// Mitsubishi GX Developer project: Пресс 70 крышка(алгоритм аварии при невыбросе крышки)   PLC: Q04UDEH

PROGRAM MAIN
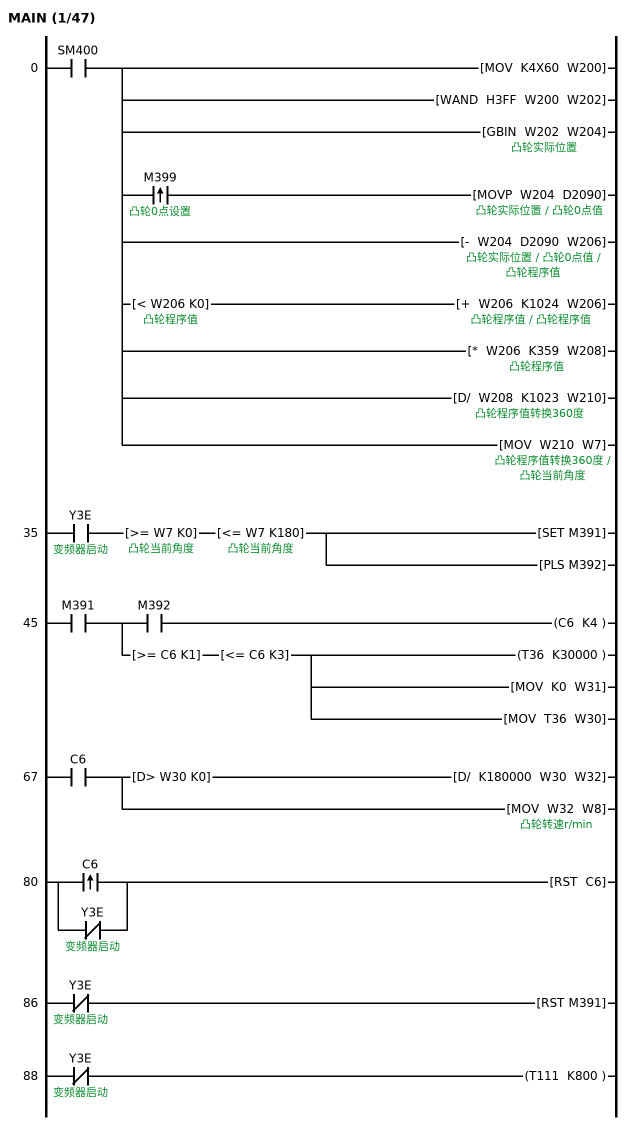
0     LD      SM400
      MOV     K4X60 W200  ; 绝地值编码器1
      WAND    H3FF W200 W202
      GBIN    W202 W204  ; 凸轮实际位置
      MPS
      ANDP    M399  ; 凸轮0点设置
      MOVP    W204 D2090  ; 凸轮0点值
      MPP
      -       W204 D2090 W206  ; 凸轮程序值
      MPS
      AND<    W206 K0  ; 凸轮程序值
      +       W206 K1024 W206
      MPP
      *       W206 K359 W208
      D/      W208 K1023 W210  ; 凸轮程序值转换360度
      MOV     W210 W7  ; 凸轮当前角度
35    LD      Y3E  ; 变频器启动
      AND>=   W7 K0  ; 凸轮当前角度
      AND<=   W7 K180  ; 凸轮当前角度
      SET     M391
      PLS     M392
45    LD      M391
      MPS
      AND     M392
      OUT     C6 K4
      MPP
      AND>=   C6 K1
      AND<=   C6 K3
      OUTH    T36 K30000
      MOV     K0 W31
      MOV     T36 W30
67    LD      C6
      MPS
      ANDD>   W30 K0
      D/      K180000 W30 W32
      MPP
      MOV     W32 W8  ; 凸轮转速r/min
80    LDP     C6
      ORI     Y3E  ; 变频器启动
      RST     C6
86    LDI     Y3E  ; 变频器启动
      RST     M391
88    LDI     Y3E  ; 变频器启动
      OUT     T111 K800
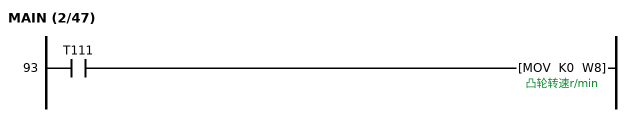
93    LD      T111
      MOV     K0 W8
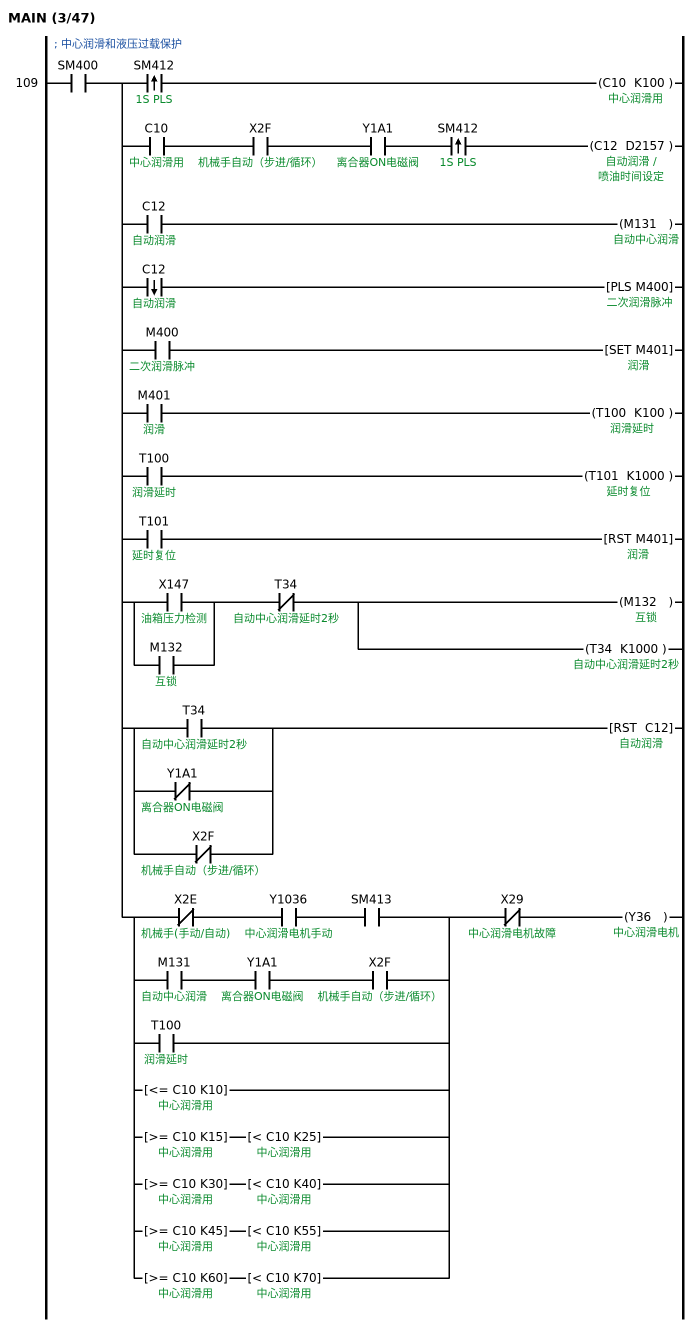
; 中心润滑和液压过载保护
109   LD      SM400
      MPS
      ANDP    SM412  ; 1S PLS
      OUT     C10 K100  ; 中心润滑用
      MRD
      AND     C10  ; 中心润滑用
      AND     X2F  ; 机械手自动（步进/循环）
      AND     Y1A1  ; 离合器ON电磁阀
      ANDP    SM412  ; 1S PLS
      OUT     C12 D2157  ; 自动润滑 / 喷油时间设定
      MRD
      AND     C12  ; 自动润滑
      OUT     M131  ; 自动中心润滑
      MRD
      ANDF    C12  ; 自动润滑
      PLS     M400  ; 二次润滑脉冲
      MRD
      AND     M400  ; 二次润滑脉冲
      SET     M401  ; 润滑
      MRD
      AND     M401  ; 润滑
      OUT     T100 K100  ; 润滑延时
      MRD
      AND     T100  ; 润滑延时
      OUT     T101 K1000  ; 延时复位
      MRD
      AND     T101  ; 延时复位
      RST     M401  ; 润滑
      MRD
      LD      X147  ; 油箱压力检测
      OR      M132  ; 互锁
      ANB
      ANI     T34  ; 自动中心润滑延时2秒
      OUT     M132  ; 互锁
      OUT     T34 K1000  ; 自动中心润滑延时2秒
      MRD
      LD      T34  ; 自动中心润滑延时2秒
      ORI     Y1A1  ; 离合器ON电磁阀
      ORI     X2F  ; 机械手自动（步进/循环）
      ANB
      RST     C12  ; 自动润滑
      MPP
      LDI     X2E  ; 机械手(手动/自动)
      AND     Y1036  ; 中心润滑电机手动
      AND     SM413
      LD      M131  ; 自动中心润滑
      AND     Y1A1  ; 离合器ON电磁阀
      AND     X2F  ; 机械手自动（步进/循环）
      ORB
      OR      T100  ; 润滑延时
      OR<=    C10 K10  ; 中心润滑用
      LD>=    C10 K15  ; 中心润滑用
      AND<    C10 K25  ; 中心润滑用
      ORB
      LD>=    C10 K30  ; 中心润滑用
      AND<    C10 K40  ; 中心润滑用
      ORB
      LD>=    C10 K45  ; 中心润滑用
      AND<    C10 K55  ; 中心润滑用
      ORB
      LD>=    C10 K60  ; 中心润滑用
      AND<    C10 K70  ; 中心润滑用
      ORB
      ANB
      ANI     X29  ; 中心润滑电机故障
      OUT     Y36  ; 中心润滑电机
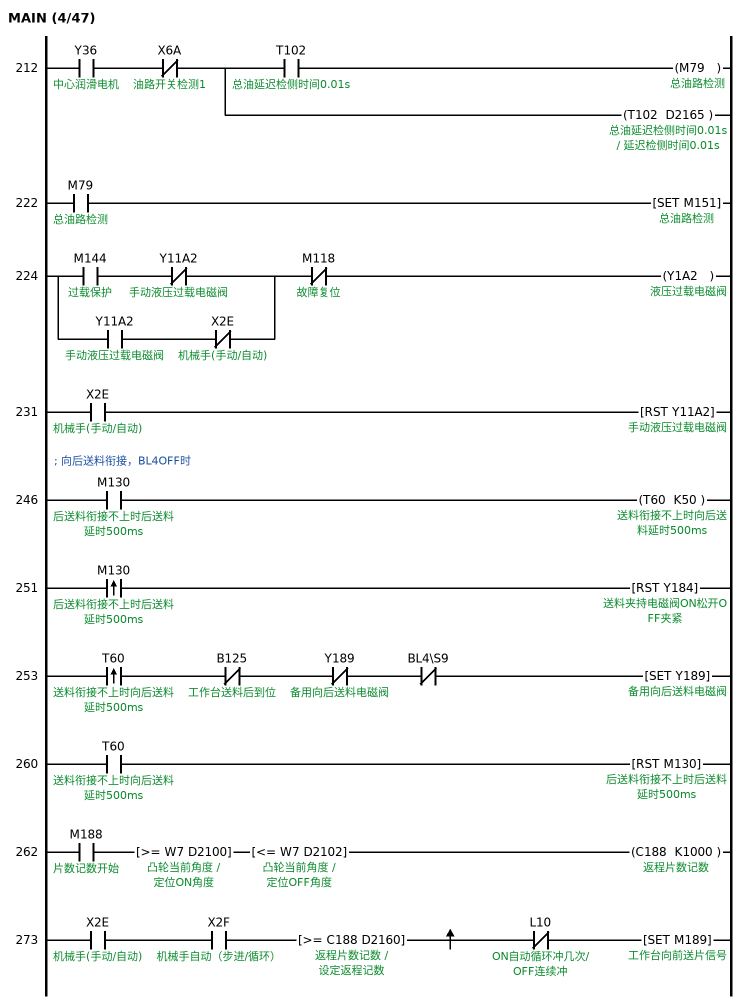
212   LD      Y36  ; 中心润滑电机
      ANI     X6A  ; 油路开关检测1
      MPS
      AND     T102  ; 总油延迟检侧时间0.01s
      OUT     M79  ; 总油路检测
      MPP
      OUT     T102 D2165  ; 总油延迟检侧时间0.01s / 延迟检侧时间0.01s
222   LD      M79  ; 总油路检测
      SET     M151  ; 总油路检测
224   LD      M144  ; 过载保护
      ANI     Y11A2  ; 手动液压过载电磁阀
      LD      Y11A2  ; 手动液压过载电磁阀
      ANI     X2E  ; 机械手(手动/自动)
      ORB
      ANI     M118  ; 故障复位
      OUT     Y1A2  ; 液压过载电磁阀
231   LD      X2E  ; 机械手(手动/自动)
      RST     Y11A2  ; 手动液压过载电磁阀
; 向后送料衔接，BL4OFF时
246   LD      M130  ; 后送料衔接不上时后送料延时500ms
      OUT     T60 K50  ; 送料衔接不上时向后送料延时500ms
251   LDP     M130  ; 后送料衔接不上时后送料延时500ms
      RST     Y184  ; 送料夹持电磁阀ON松开OFF夹紧
253   LDP     T60  ; 送料衔接不上时向后送料延时500ms
      ANI     B125  ; 工作台送料后到位
      ANI     Y189  ; 备用向后送料电磁阀
      ANI     BL4\S9
      SET     Y189  ; 备用向后送料电磁阀
260   LD      T60  ; 送料衔接不上时向后送料延时500ms
      RST     M130  ; 后送料衔接不上时后送料延时500ms
262   LD      M188  ; 片数记数开始
      AND>=   W7 D2100  ; 凸轮当前角度 / 定位ON角度
      AND<=   W7 D2102  ; 凸轮当前角度 / 定位OFF角度
      OUT     C188 K1000  ; 返程片数记数
273   LD      X2E  ; 机械手(手动/自动)
      AND     X2F  ; 机械手自动（步进/循环）
      AND>=   C188 D2160  ; 返程片数记数 / 设定返程记数
      MEP
      ANI     L10  ; ON自动循环冲几次/OFF连续冲
      SET     M189  ; 工作台向前送片信号
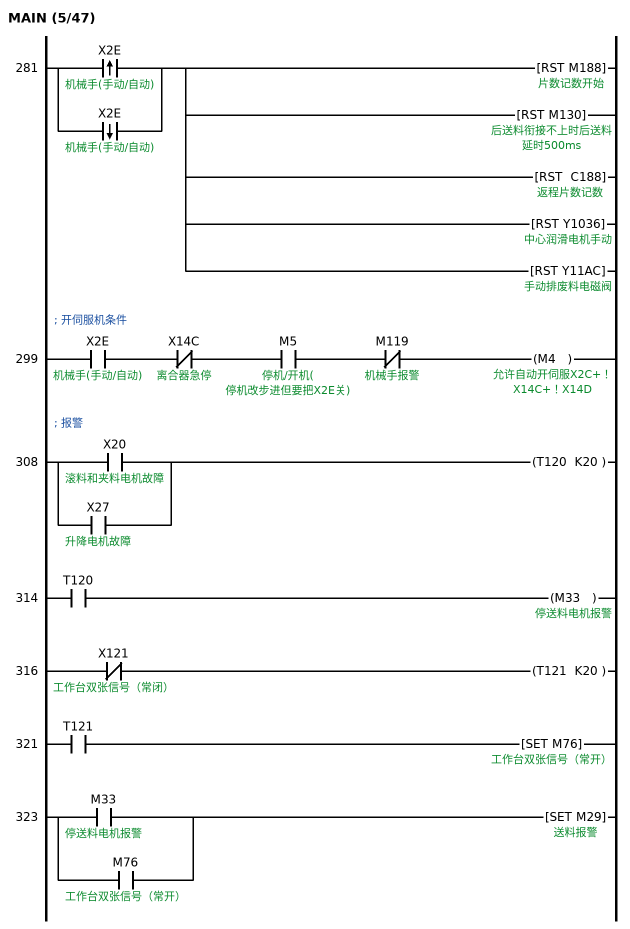
281   LDP     X2E  ; 机械手(手动/自动)
      ORF     X2E  ; 机械手(手动/自动)
      RST     M188  ; 片数记数开始
      RST     M130  ; 后送料衔接不上时后送料延时500ms
      RST     C188  ; 返程片数记数
      RST     Y1036  ; 中心润滑电机手动
      RST     Y11AC  ; 手动排废料电磁阀
; 开伺服机条件
299   LD      X2E  ; 机械手(手动/自动)
      ANI     X14C  ; 离合器急停
      AND     M5  ; 停机/开机(停机改步进但要把X2E关)
      ANI     M119  ; 机械手报警
      OUT     M4  ; 允许自动开伺服X2C+！X14C+！X14D
; 报警
308   LD      X20  ; 滚料和夹料电机故障
      OR      X27  ; 升降电机故障
      OUT     T120 K20
314   LD      T120
      OUT     M33  ; 停送料电机报警
316   LDI     X121  ; 工作台双张信号（常闭）
      OUT     T121 K20
321   LD      T121
      SET     M76  ; 工作台双张信号（常开）
323   LD      M33  ; 停送料电机报警
      OR      M76  ; 工作台双张信号（常开）
      SET     M29  ; 送料报警
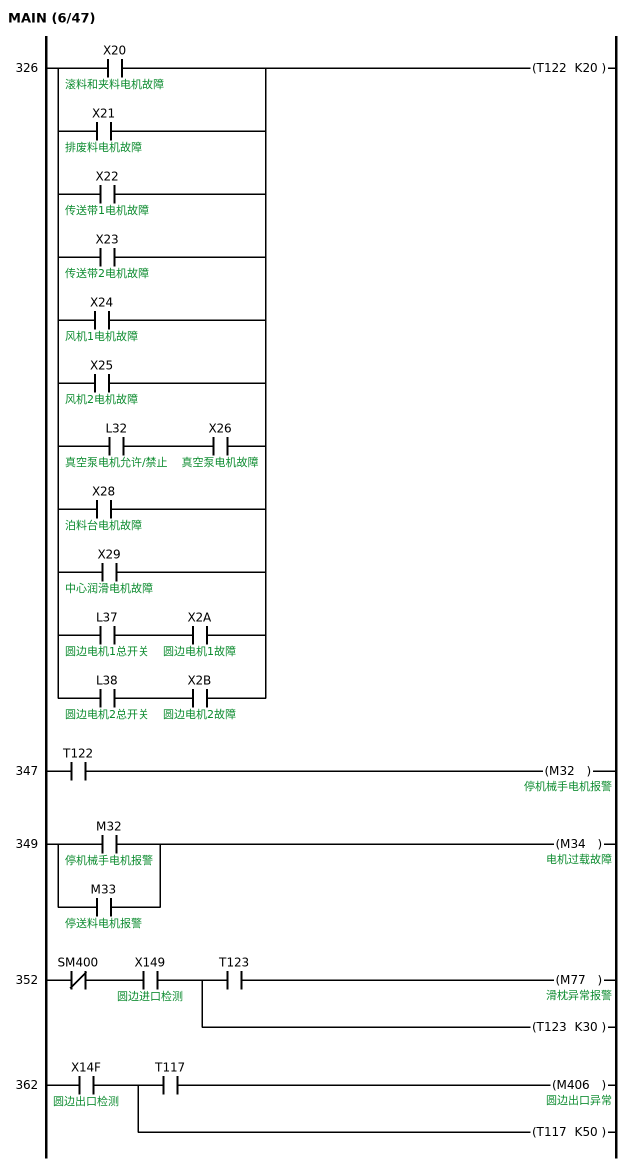
326   LD      X20  ; 滚料和夹料电机故障
      OR      X21  ; 排废料电机故障
      OR      X22  ; 传送带1电机故障
      OR      X23  ; 传送带2电机故障
      OR      X24  ; 风机1电机故障
      OR      X25  ; 风机2电机故障
      LD      L32  ; 真空泵电机允许/禁止
      AND     X26  ; 真空泵电机故障
      ORB
      OR      X28  ; 泊料台电机故障
      OR      X29  ; 中心润滑电机故障
      LD      L37  ; 圆边电机1总开关
      AND     X2A  ; 圆边电机1故障
      ORB
      LD      L38  ; 圆边电机2总开关
      AND     X2B  ; 圆边电机2故障
      ORB
      OUT     T122 K20
347   LD      T122
      OUT     M32  ; 停机械手电机报警
349   LD      M32  ; 停机械手电机报警
      OR      M33  ; 停送料电机报警
      OUT     M34  ; 电机过载故障
352   LDI     SM400
      AND     X149  ; 圆边进口检测
      MPS
      AND     T123
      OUT     M77  ; 滑枕异常报警
      MPP
      OUT     T123 K30
362   LD      X14F  ; 圆边出口检测
      MPS
      AND     T117
      OUT     M406  ; 圆边出口异常
      MPP
      OUT     T117 K50
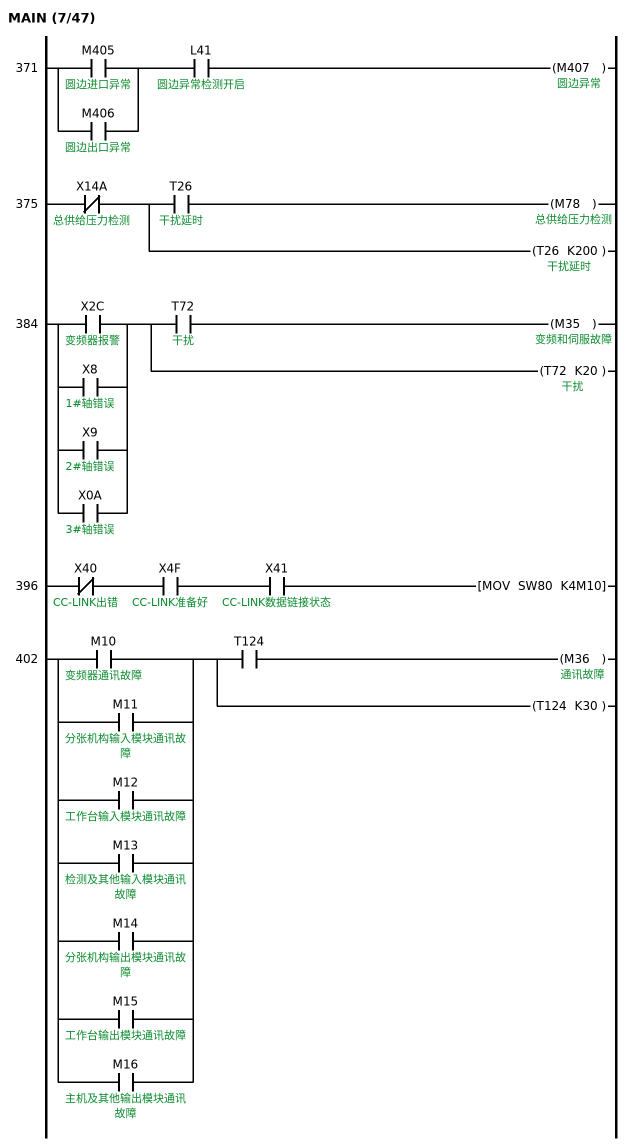
371   LD      M405  ; 圆边进口异常
      OR      M406  ; 圆边出口异常
      AND     L41  ; 圆边异常检测开启
      OUT     M407  ; 圆边异常
375   LDI     X14A  ; 总供给压力检测
      MPS
      AND     T26  ; 干扰延时
      OUT     M78  ; 总供给压力检测
      MPP
      OUT     T26 K200  ; 干扰延时
384   LD      X2C  ; 变频器报警
      OR      X8  ; 1#轴错误
      OR      X9  ; 2#轴错误
      OR      X0A  ; 3#轴错误
      MPS
      AND     T72  ; 干扰
      OUT     M35  ; 变频和伺服故障
      MPP
      OUT     T72 K20  ; 干扰
396   LDI     X40  ; CC-LINK出错
      AND     X4F  ; CC-LINK准备好
      AND     X41  ; CC-LINK数据链接状态
      MOV     SW80 K4M10  ; 变频器通讯故障
402   LD      M10  ; 变频器通讯故障
      OR      M11  ; 分张机构输入模块通讯故障
      OR      M12  ; 工作台输入模块通讯故障
      OR      M13  ; 检测及其他输入模块通讯故障
      OR      M14  ; 分张机构输出模块通讯故障
      OR      M15  ; 工作台输出模块通讯故障
      OR      M16  ; 主机及其他输出模块通讯故障
      MPS
      AND     T124
      OUT     M36  ; 通讯故障
      MPP
      OUT     T124 K30
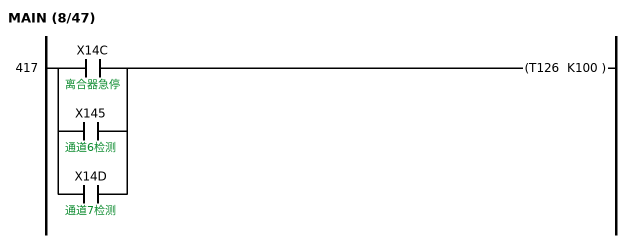
417   LD      X14C  ; 离合器急停
      OR      X145  ; 通道6检测
      OR      X14D  ; 通道7检测
      OUTH    T126 K100
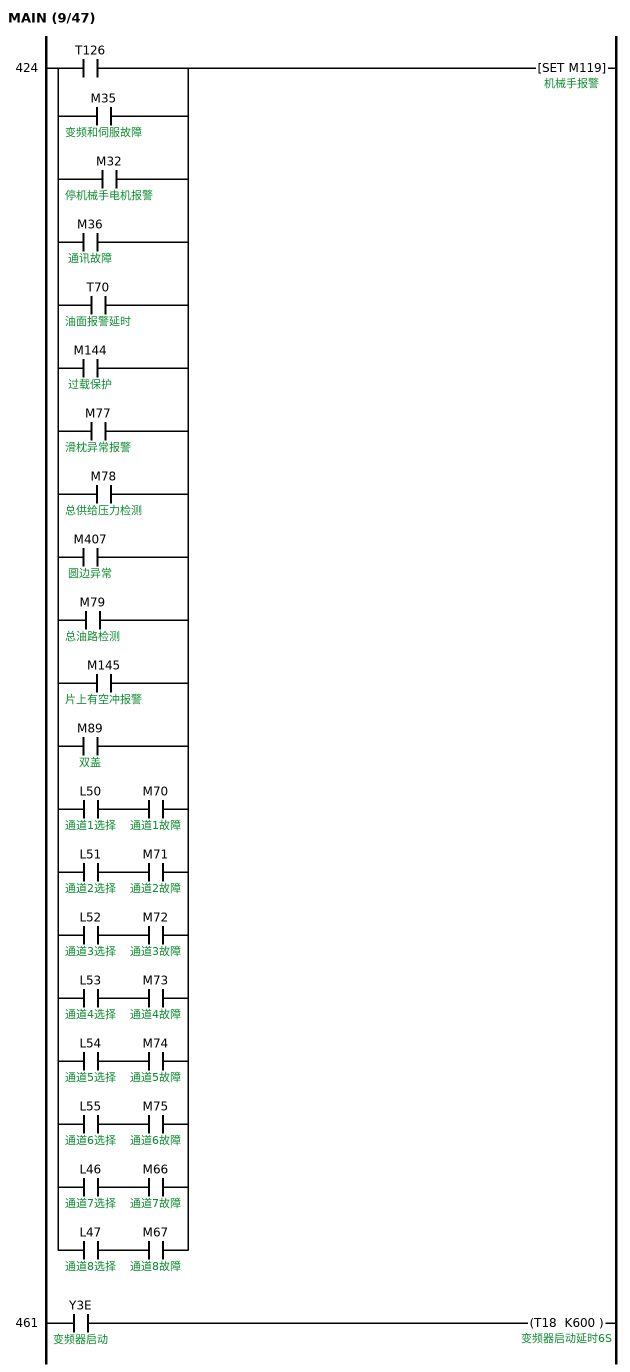
424   LD      T126
      OR      M35  ; 变频和伺服故障
      OR      M32  ; 停机械手电机报警
      OR      M36  ; 通讯故障
      OR      T70  ; 油面报警延时
      OR      M144  ; 过载保护
      OR      M77  ; 滑枕异常报警
      OR      M78  ; 总供给压力检测
      OR      M407  ; 圆边异常
      OR      M79  ; 总油路检测
      OR      M145  ; 片上有空冲报警
      OR      M89  ; 双盖
      LD      L50  ; 通道1选择
      AND     M70  ; 通道1故障
      ORB
      LD      L51  ; 通道2选择
      AND     M71  ; 通道2故障
      ORB
      LD      L52  ; 通道3选择
      AND     M72  ; 通道3故障
      ORB
      LD      L53  ; 通道4选择
      AND     M73  ; 通道4故障
      ORB
      LD      L54  ; 通道5选择
      AND     M74  ; 通道5故障
      ORB
      LD      L55  ; 通道6选择
      AND     M75  ; 通道6故障
      ORB
      LD      L46  ; 通道7选择
      AND     M66  ; 通道7故障
      ORB
      LD      L47  ; 通道8选择
      AND     M67  ; 通道8故障
      ORB
      SET     M119  ; 机械手报警
461   LD      Y3E  ; 变频器启动
      OUT     T18 K600  ; 变频器启动延时6S
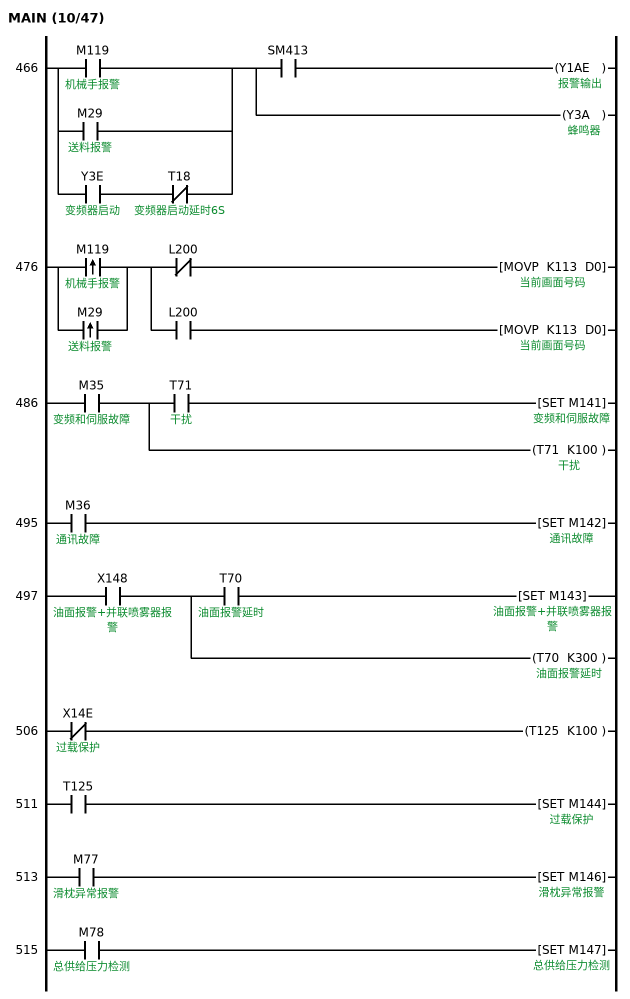
466   LD      M119  ; 机械手报警
      OR      M29  ; 送料报警
      LD      Y3E  ; 变频器启动
      ANI     T18  ; 变频器启动延时6S
      ORB
      MPS
      AND     SM413
      OUT     Y1AE  ; 报警输出
      MPP
      OUT     Y3A  ; 蜂鸣器
476   LDP     M119  ; 机械手报警
      ORP     M29  ; 送料报警
      MPS
      ANI     L200
      MOVP    K113 D0  ; 当前画面号码
      MPP
      AND     L200
      MOVP    K113 D0
486   LD      M35  ; 变频和伺服故障
      MPS
      AND     T71  ; 干扰
      SET     M141  ; 变频和伺服故障
      MPP
      OUT     T71 K100  ; 干扰
495   LD      M36  ; 通讯故障
      SET     M142  ; 通讯故障
497   LD      X148  ; 油面报警+并联喷雾器报警
      MPS
      AND     T70  ; 油面报警延时
      SET     M143  ; 油面报警+并联喷雾器报警
      MPP
      OUT     T70 K300  ; 油面报警延时
506   LDI     X14E  ; 过载保护
      OUTH    T125 K100
511   LD      T125
      SET     M144  ; 过载保护
513   LD      M77  ; 滑枕异常报警
      SET     M146  ; 滑枕异常报警
515   LD      M78  ; 总供给压力检测
      SET     M147  ; 总供给压力检测
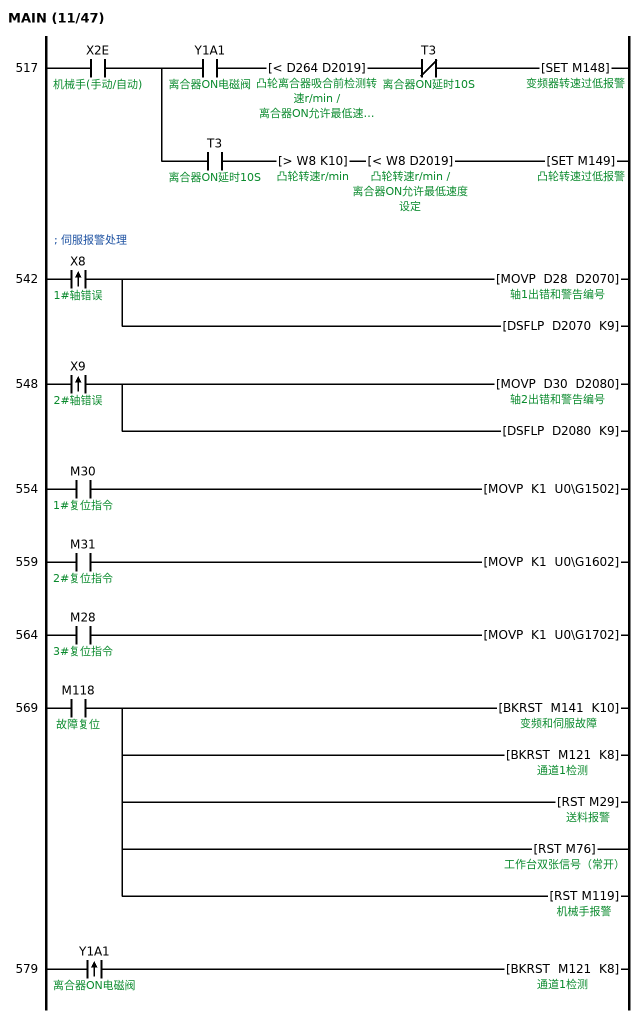
517   LD      X2E  ; 机械手(手动/自动)
      MPS
      AND     Y1A1  ; 离合器ON电磁阀
      AND<    D264 D2019  ; 凸轮离合器吸合前检测转速r/min / 离合器ON允许最低速度设定
      ANI     T3  ; 离合器ON延时10S
      SET     M148  ; 变频器转速过低报警
      MPP
      AND     T3  ; 离合器ON延时10S
      AND>    W8 K10  ; 凸轮转速r/min
      AND<    W8 D2019  ; 凸轮转速r/min / 离合器ON允许最低速度设定
      SET     M149  ; 凸轮转速过低报警
; 伺服报警处理
542   LDP     X8  ; 1#轴错误
      MOVP    D28 D2070  ; 轴1出错和警告编号
      DSFLP   D2070 K9
548   LDP     X9  ; 2#轴错误
      MOVP    D30 D2080  ; 轴2出错和警告编号
      DSFLP   D2080 K9
554   LD      M30  ; 1#复位指令
      MOVP    K1 U0\G1502
559   LD      M31  ; 2#复位指令
      MOVP    K1 U0\G1602
564   LD      M28  ; 3#复位指令
      MOVP    K1 U0\G1702
569   LD      M118  ; 故障复位
      BKRST   M141 K10
      BKRST   M121 K8  ; 通道1检测
      RST     M29  ; 送料报警
      RST     M76  ; 工作台双张信号（常开）
      RST     M119  ; 机械手报警
579   LDP     Y1A1  ; 离合器ON电磁阀
      BKRST   M121 K8
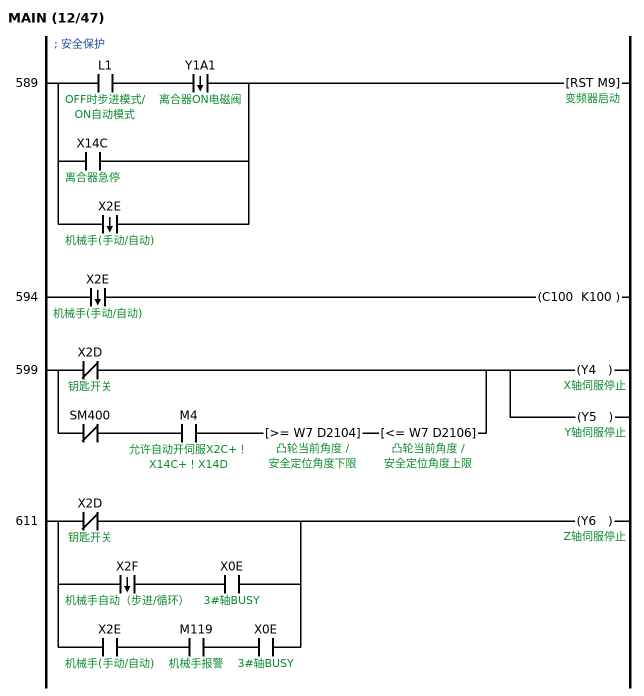
; 安全保护
589   LD      L1  ; OFF时步进模式/ON自动模式
      ANDF    Y1A1  ; 离合器ON电磁阀
      OR      X14C  ; 离合器急停
      ORF     X2E  ; 机械手(手动/自动)
      RST     M9  ; 变频器启动
594   LDF     X2E  ; 机械手(手动/自动)
      OUT     C100 K100
599   LDI     X2D  ; 钥匙开关
      LDI     SM400
      AND     M4  ; 允许自动开伺服X2C+！X14C+！X14D
      AND>=   W7 D2104  ; 凸轮当前角度 / 安全定位角度下限
      AND<=   W7 D2106  ; 凸轮当前角度 / 安全定位角度上限
      ORB
      OUT     Y4  ; X轴伺服停止
      OUT     Y5  ; Y轴伺服停止
611   LDI     X2D  ; 钥匙开关
      LDF     X2F  ; 机械手自动（步进/循环）
      AND     X0E  ; 3#轴BUSY
      ORB
      LD      X2E  ; 机械手(手动/自动)
      AND     M119  ; 机械手报警
      AND     X0E  ; 3#轴BUSY
      ORB
      OUT     Y6  ; Z轴伺服停止
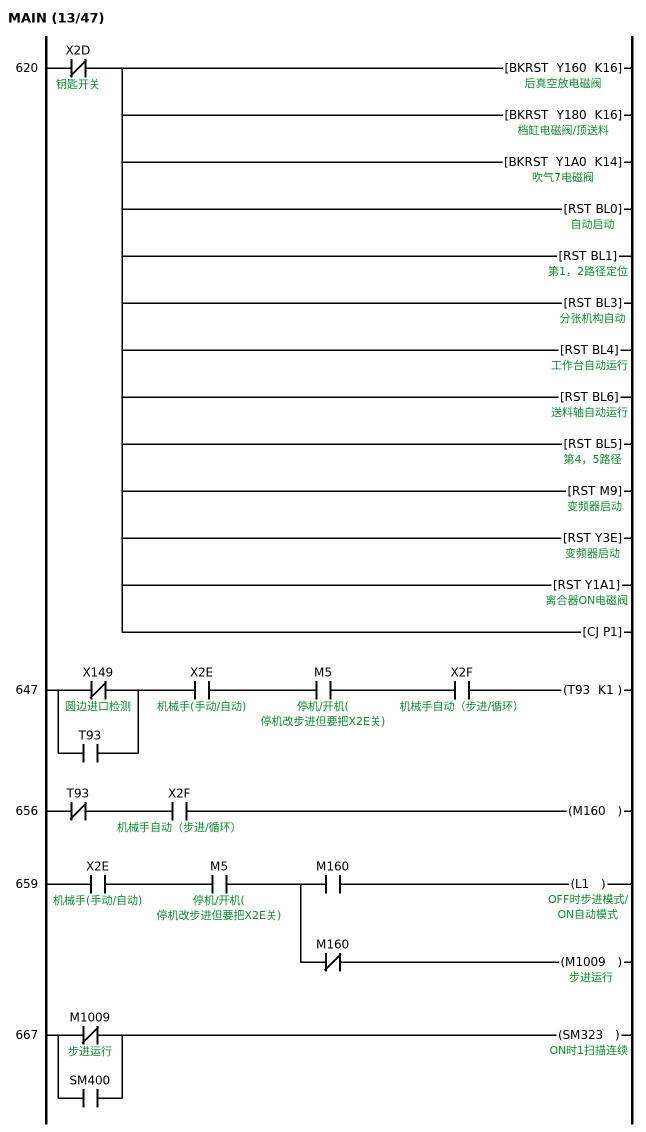
620   LDI     X2D  ; 钥匙开关
      BKRST   Y160 K16  ; 后真空放电磁阀
      BKRST   Y180 K16  ; 档缸电磁阀/顶送料
      BKRST   Y1A0 K14  ; 吹气7电磁阀
      RST     BL0  ; 自动启动
      RST     BL1  ; 第1，2路径定位
      RST     BL3  ; 分张机构自动
      RST     BL4  ; 工作台自动运行
      RST     BL6  ; 送料轴自动运行
      RST     BL5  ; 第4，5路径
      RST     M9  ; 变频器启动
      RST     Y3E  ; 变频器启动
      RST     Y1A1  ; 离合器ON电磁阀
      CJ      P1
647   LDI     X149  ; 圆边进口检测
      OR      T93
      AND     X2E  ; 机械手(手动/自动)
      AND     M5  ; 停机/开机(停机改步进但要把X2E关)
      AND     X2F  ; 机械手自动（步进/循环）
      OUT     T93 K1
656   LDI     T93
      AND     X2F  ; 机械手自动（步进/循环）
      OUT     M160
659   LD      X2E  ; 机械手(手动/自动)
      AND     M5  ; 停机/开机(停机改步进但要把X2E关)
      MPS
      AND     M160
      OUT     L1  ; OFF时步进模式/ON自动模式
      MPP
      ANI     M160
      OUT     M1009  ; 步进运行
667   LDI     M1009  ; 步进运行
      OR      SM400
      OUT     SM323  ; ON时1扫描连续
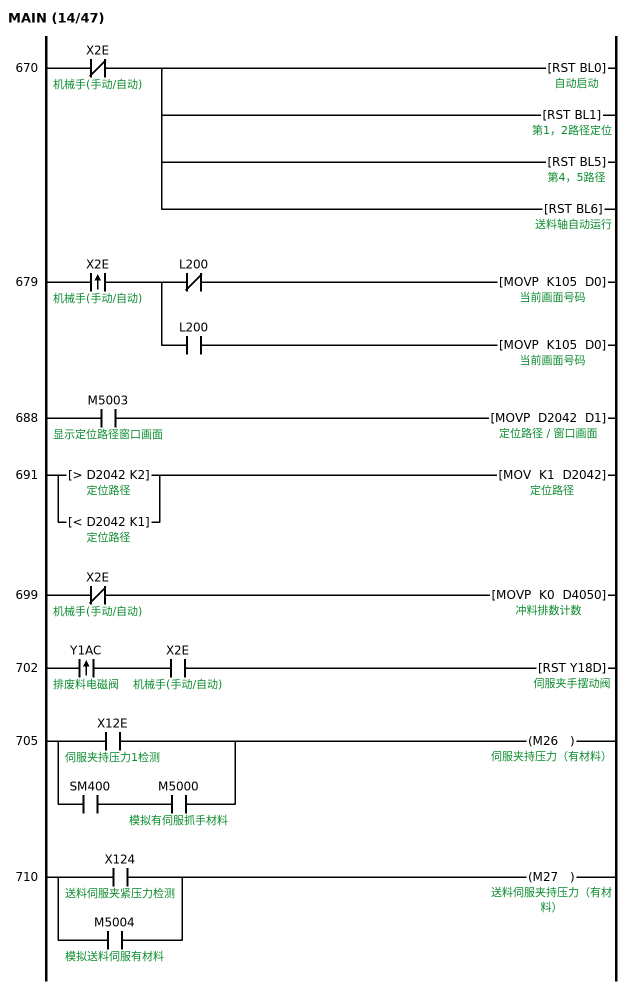
670   LDI     X2E  ; 机械手(手动/自动)
      RST     BL0  ; 自动启动
      RST     BL1  ; 第1，2路径定位
      RST     BL5  ; 第4，5路径
      RST     BL6  ; 送料轴自动运行
679   LDP     X2E  ; 机械手(手动/自动)
      MPS
      ANI     L200
      MOVP    K105 D0
      MPP
      AND     L200
      MOVP    K105 D0
688   LD      M5003  ; 显示定位路径窗口画面
      MOVP    D2042 D1  ; 定位路径 / 窗口画面
691   LD>     D2042 K2  ; 定位路径
      OR<     D2042 K1  ; 定位路径
      MOV     K1 D2042
699   LDI     X2E  ; 机械手(手动/自动)
      MOVP    K0 D4050  ; 冲料排数计数
702   LDP     Y1AC  ; 排废料电磁阀
      AND     X2E  ; 机械手(手动/自动)
      RST     Y18D  ; 伺服夹手摆动阀
705   LD      X12E  ; 伺服夹持压力1检测
      LD      SM400
      AND     M5000  ; 模拟有伺服抓手材料
      ORB
      OUT     M26  ; 伺服夹持压力（有材料）
710   LD      X124  ; 送料伺服夹紧压力检测
      OR      M5004  ; 模拟送料伺服有材料
      OUT     M27  ; 送料伺服夹持压力（有材料）
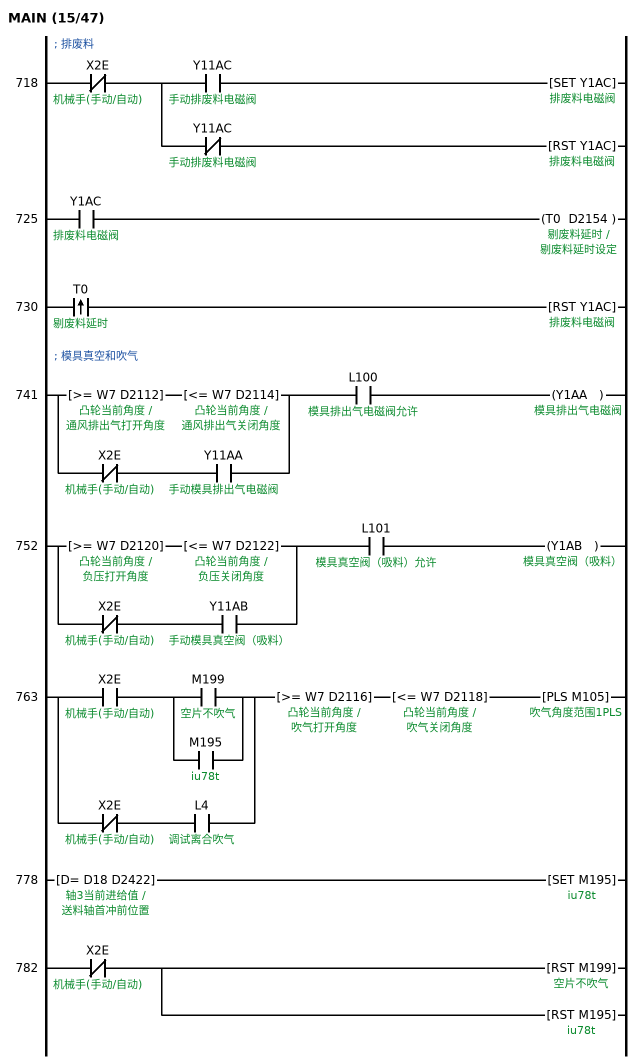
; 排废料
718   LDI     X2E  ; 机械手(手动/自动)
      MPS
      AND     Y11AC  ; 手动排废料电磁阀
      SET     Y1AC  ; 排废料电磁阀
      MPP
      ANI     Y11AC  ; 手动排废料电磁阀
      RST     Y1AC  ; 排废料电磁阀
725   LD      Y1AC  ; 排废料电磁阀
      OUTH    T0 D2154  ; 剔废料延时 / 剔废料延时设定
730   LDP     T0  ; 剔废料延时
      RST     Y1AC  ; 排废料电磁阀
; 模具真空和吹气
741   LD>=    W7 D2112  ; 凸轮当前角度 / 通风排出气打开角度
      AND<=   W7 D2114  ; 凸轮当前角度 / 通风排出气关闭角度
      LDI     X2E  ; 机械手(手动/自动)
      AND     Y11AA  ; 手动模具排出气电磁阀
      ORB
      AND     L100  ; 模具排出气电磁阀允许
      OUT     Y1AA  ; 模具排出气电磁阀
752   LD>=    W7 D2120  ; 凸轮当前角度 / 负压打开角度
      AND<=   W7 D2122  ; 凸轮当前角度 / 负压关闭角度
      LDI     X2E  ; 机械手(手动/自动)
      AND     Y11AB  ; 手动模具真空阀（吸料）
      ORB
      AND     L101  ; 模具真空阀（吸料）允许
      OUT     Y1AB  ; 模具真空阀（吸料）
763   LD      X2E  ; 机械手(手动/自动)
      LD      M199  ; 空片不吹气
      OR      M195  ; iu78t
      ANB
      LDI     X2E  ; 机械手(手动/自动)
      AND     L4  ; 调试离合吹气
      ORB
      AND>=   W7 D2116  ; 凸轮当前角度 / 吹气打开角度
      AND<=   W7 D2118  ; 凸轮当前角度 / 吹气关闭角度
      PLS     M105  ; 吹气角度范围1PLS
778   LDD=    D18 D2422  ; 轴3当前进给值 / 送料轴首冲前位置
      SET     M195  ; iu78t
782   LDI     X2E  ; 机械手(手动/自动)
      RST     M199  ; 空片不吹气
      RST     M195  ; iu78t
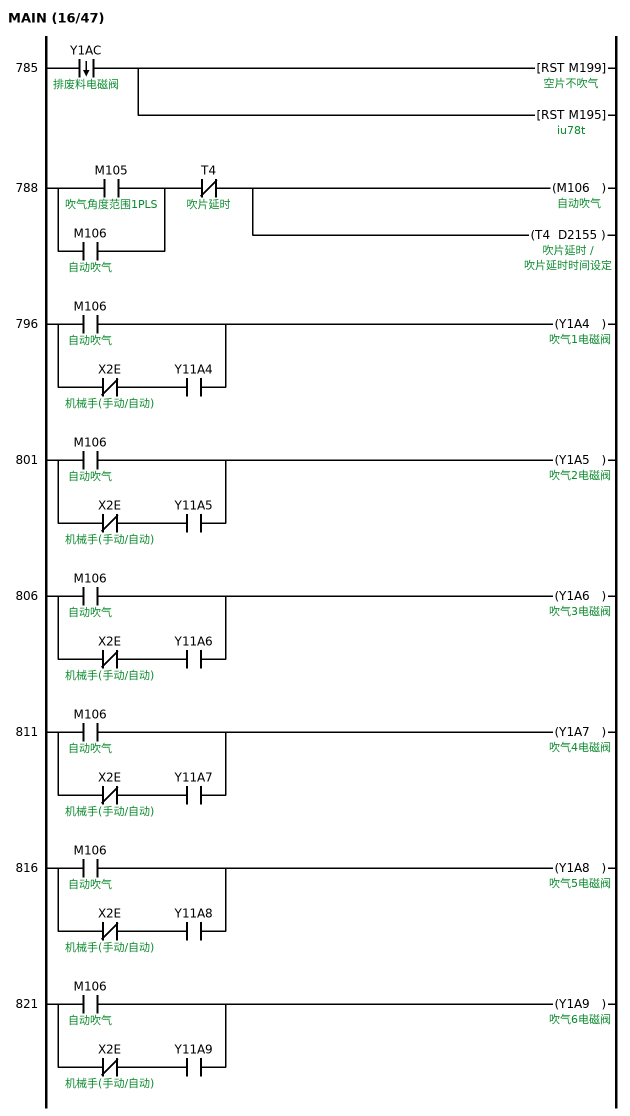
785   LDF     Y1AC  ; 排废料电磁阀
      RST     M199  ; 空片不吹气
      RST     M195  ; iu78t
788   LD      M105  ; 吹气角度范围1PLS
      OR      M106  ; 自动吹气
      ANI     T4  ; 吹片延时
      OUT     M106  ; 自动吹气
      OUTH    T4 D2155  ; 吹片延时 / 吹片延时时间设定
796   LD      M106  ; 自动吹气
      LDI     X2E  ; 机械手(手动/自动)
      AND     Y11A4
      ORB
      OUT     Y1A4  ; 吹气1电磁阀
801   LD      M106  ; 自动吹气
      LDI     X2E  ; 机械手(手动/自动)
      AND     Y11A5
      ORB
      OUT     Y1A5  ; 吹气2电磁阀
806   LD      M106  ; 自动吹气
      LDI     X2E  ; 机械手(手动/自动)
      AND     Y11A6
      ORB
      OUT     Y1A6  ; 吹气3电磁阀
811   LD      M106  ; 自动吹气
      LDI     X2E  ; 机械手(手动/自动)
      AND     Y11A7
      ORB
      OUT     Y1A7  ; 吹气4电磁阀
816   LD      M106  ; 自动吹气
      LDI     X2E  ; 机械手(手动/自动)
      AND     Y11A8
      ORB
      OUT     Y1A8  ; 吹气5电磁阀
821   LD      M106  ; 自动吹气
      LDI     X2E  ; 机械手(手动/自动)
      AND     Y11A9
      ORB
      OUT     Y1A9  ; 吹气6电磁阀
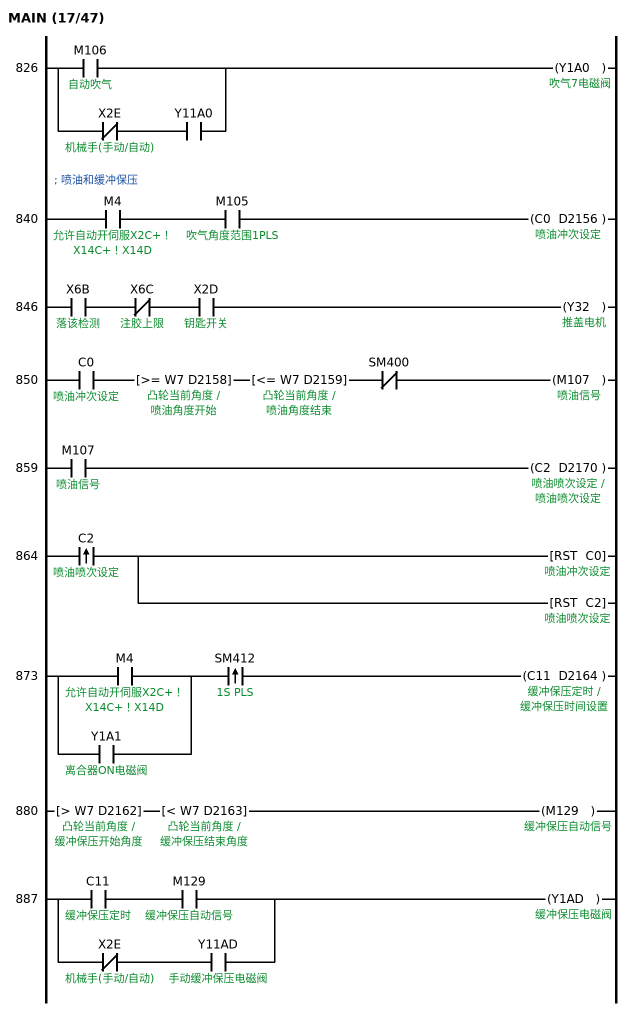
826   LD      M106  ; 自动吹气
      LDI     X2E  ; 机械手(手动/自动)
      AND     Y11A0
      ORB
      OUT     Y1A0  ; 吹气7电磁阀
; 喷油和缓冲保压
840   LD      M4  ; 允许自动开伺服X2C+！X14C+！X14D
      AND     M105  ; 吹气角度范围1PLS
      OUT     C0 D2156  ; 喷油冲次设定
846   LD      X6B  ; 落该检测
      ANI     X6C  ; 注胶上限
      AND     X2D  ; 钥匙开关
      OUT     Y32  ; 推盖电机
850   LD      C0  ; 喷油冲次设定
      AND>=   W7 D2158  ; 凸轮当前角度 / 喷油角度开始
      AND<=   W7 D2159  ; 凸轮当前角度 / 喷油角度结束
      ANI     SM400
      OUT     M107  ; 喷油信号
859   LD      M107  ; 喷油信号
      OUT     C2 D2170  ; 喷油喷次设定 / 喷油喷次设定
864   LDP     C2  ; 喷油喷次设定
      RST     C0  ; 喷油冲次设定
      RST     C2  ; 喷油喷次设定
873   LD      M4  ; 允许自动开伺服X2C+！X14C+！X14D
      OR      Y1A1  ; 离合器ON电磁阀
      ANDP    SM412  ; 1S PLS
      OUT     C11 D2164  ; 缓冲保压定时 / 缓冲保压时间设置
880   LD>     W7 D2162  ; 凸轮当前角度 / 缓冲保压开始角度
      AND<    W7 D2163  ; 凸轮当前角度 / 缓冲保压结束角度
      OUT     M129  ; 缓冲保压自动信号
887   LD      C11  ; 缓冲保压定时
      AND     M129  ; 缓冲保压自动信号
      LDI     X2E  ; 机械手(手动/自动)
      AND     Y11AD  ; 手动缓冲保压电磁阀
      ORB
      OUT     Y1AD  ; 缓冲保压电磁阀
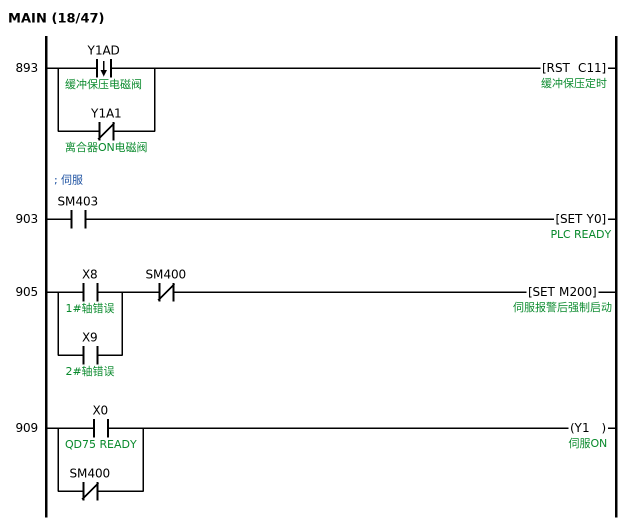
893   LDF     Y1AD  ; 缓冲保压电磁阀
      ORI     Y1A1  ; 离合器ON电磁阀
      RST     C11  ; 缓冲保压定时
; 伺服
903   LD      SM403
      SET     Y0  ; PLC READY
905   LD      X8  ; 1#轴错误
      OR      X9  ; 2#轴错误
      ANI     SM400
      SET     M200  ; 伺服报警后强制启动
909   LD      X0  ; QD75 READY
      ORI     SM400
      OUT     Y1  ; 伺服ON
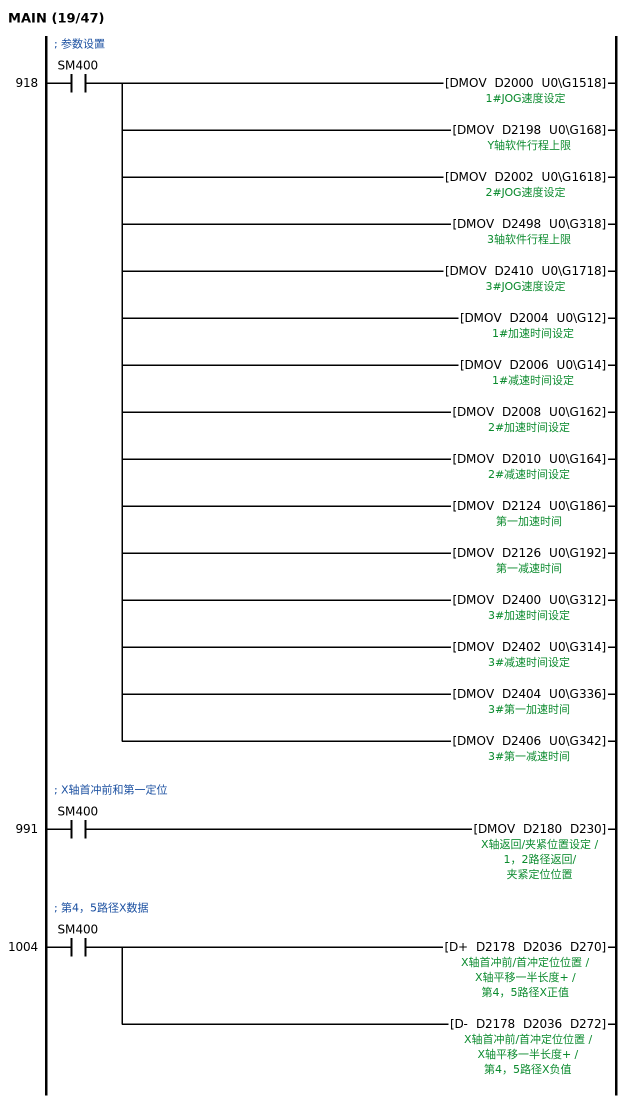
; 参数设置
918   LD      SM400
      DMOV    D2000 U0\G1518  ; 1#JOG速度设定
      DMOV    D2198 U0\G168  ; Y轴软件行程上限
      DMOV    D2002 U0\G1618  ; 2#JOG速度设定
      DMOV    D2498 U0\G318  ; 3轴软件行程上限
      DMOV    D2410 U0\G1718  ; 3#JOG速度设定
      DMOV    D2004 U0\G12  ; 1#加速时间设定
      DMOV    D2006 U0\G14  ; 1#减速时间设定
      DMOV    D2008 U0\G162  ; 2#加速时间设定
      DMOV    D2010 U0\G164  ; 2#减速时间设定
      DMOV    D2124 U0\G186  ; 第一加速时间
      DMOV    D2126 U0\G192  ; 第一减速时间
      DMOV    D2400 U0\G312  ; 3#加速时间设定
      DMOV    D2402 U0\G314  ; 3#减速时间设定
      DMOV    D2404 U0\G336  ; 3#第一加速时间
      DMOV    D2406 U0\G342  ; 3#第一减速时间
; X轴首冲前和第一定位
991   LD      SM400
      DMOV    D2180 D230  ; X轴返回/夹紧位置设定 / 1，2路径返回/夹紧定位位置
; 第4，5路径X数据
1004  LD      SM400
      D+      D2178 D2036 D270  ; X轴首冲前/首冲定位位置 / X轴平移一半长度+ / 第4，5路径X正值
      D-      D2178 D2036 D272  ; 第4，5路径X负值
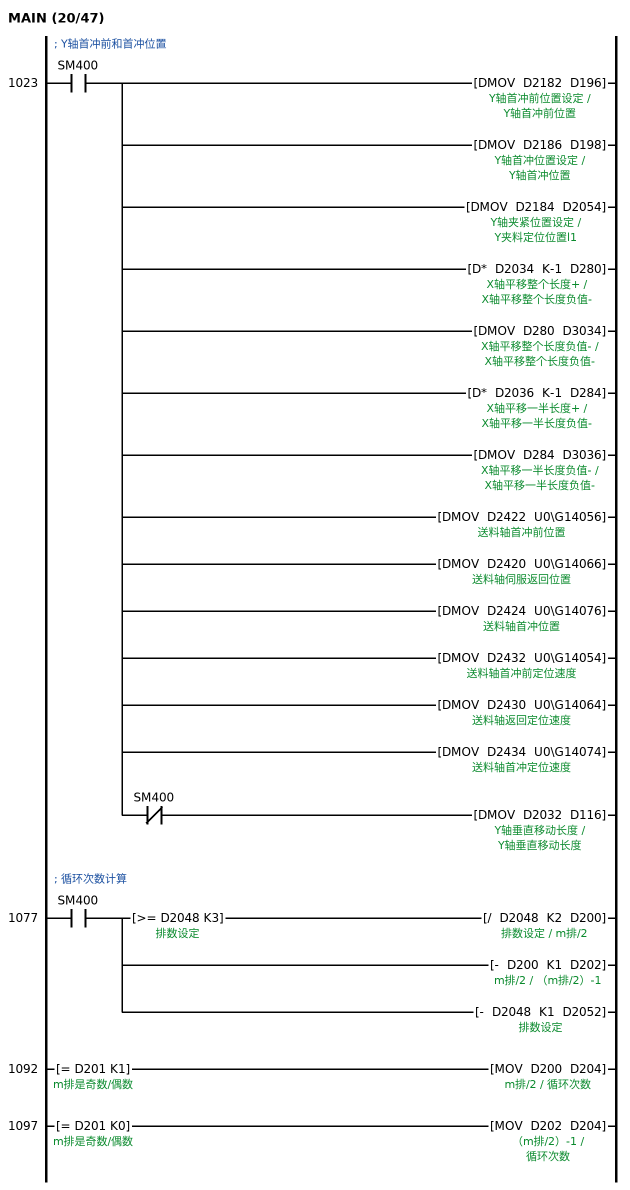
; Y轴首冲前和首冲位置
1023  LD      SM400
      DMOV    D2182 D196  ; Y轴首冲前位置设定 / Y轴首冲前位置
      DMOV    D2186 D198  ; Y轴首冲位置设定 / Y轴首冲位置
      DMOV    D2184 D2054  ; Y轴夹紧位置设定 / Y夹料定位位置l1
      D*      D2034 K-1 D280  ; X轴平移整个长度+ / X轴平移整个长度负值-
      DMOV    D280 D3034  ; X轴平移整个长度负值-
      D*      D2036 K-1 D284  ; X轴平移一半长度负值-
      DMOV    D284 D3036  ; X轴平移一半长度负值-
      DMOV    D2422 U0\G14056
      DMOV    D2420 U0\G14066  ; 送料轴伺服返回位置
      DMOV    D2424 U0\G14076  ; 送料轴首冲位置
      DMOV    D2432 U0\G14054  ; 送料轴首冲前定位速度
      DMOV    D2430 U0\G14064  ; 送料轴返回定位速度
      DMOV    D2434 U0\G14074  ; 送料轴首冲定位速度
      ANI     SM400
      DMOV    D2032 D116  ; Y轴垂直移动长度 / Y轴垂直移动长度
; 循环次数计算
1077  LD      SM400
      MPS
      AND>=   D2048 K3  ; 排数设定
      /       D2048 K2 D200  ; m排/2
      MPP
      -       D200 K1 D202  ; （m排/2）-1
      -       D2048 K1 D2052
1092  LD=     D201 K1  ; m排是奇数/偶数
      MOV     D200 D204  ; 循环次数
1097  LD=     D201 K0  ; m排是奇数/偶数
      MOV     D202 D204
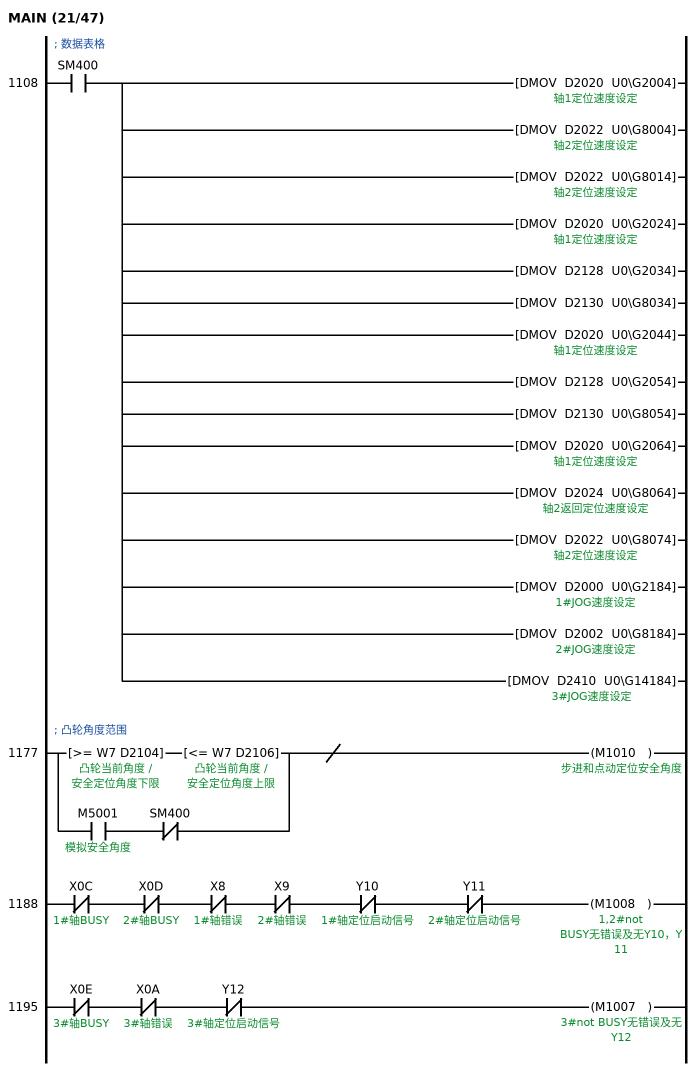
; 数据表格
1108  LD      SM400
      DMOV    D2020 U0\G2004  ; 轴1定位速度设定
      DMOV    D2022 U0\G8004  ; 轴2定位速度设定
      DMOV    D2022 U0\G8014
      DMOV    D2020 U0\G2024
      DMOV    D2128 U0\G2034
      DMOV    D2130 U0\G8034
      DMOV    D2020 U0\G2044
      DMOV    D2128 U0\G2054
      DMOV    D2130 U0\G8054
      DMOV    D2020 U0\G2064
      DMOV    D2024 U0\G8064  ; 轴2返回定位速度设定
      DMOV    D2022 U0\G8074
      DMOV    D2000 U0\G2184
      DMOV    D2002 U0\G8184
      DMOV    D2410 U0\G14184
; 凸轮角度范围
1177  LD>=    W7 D2104  ; 凸轮当前角度 / 安全定位角度下限
      AND<=   W7 D2106  ; 凸轮当前角度 / 安全定位角度上限
      LD      M5001  ; 模拟安全角度
      ANI     SM400
      ORB
      INV
      OUT     M1010  ; 步进和点动定位安全角度
1188  LDI     X0C  ; 1#轴BUSY
      ANI     X0D  ; 2#轴BUSY
      ANI     X8  ; 1#轴错误
      ANI     X9  ; 2#轴错误
      ANI     Y10  ; 1#轴定位启动信号
      ANI     Y11  ; 2#轴定位启动信号
      OUT     M1008  ; 1,2#not BUSY无错误及无Y10，Y11
1195  LDI     X0E  ; 3#轴BUSY
      ANI     X0A  ; 3#轴错误
      ANI     Y12  ; 3#轴定位启动信号
      OUT     M1007  ; 3#not BUSY无错误及无Y12
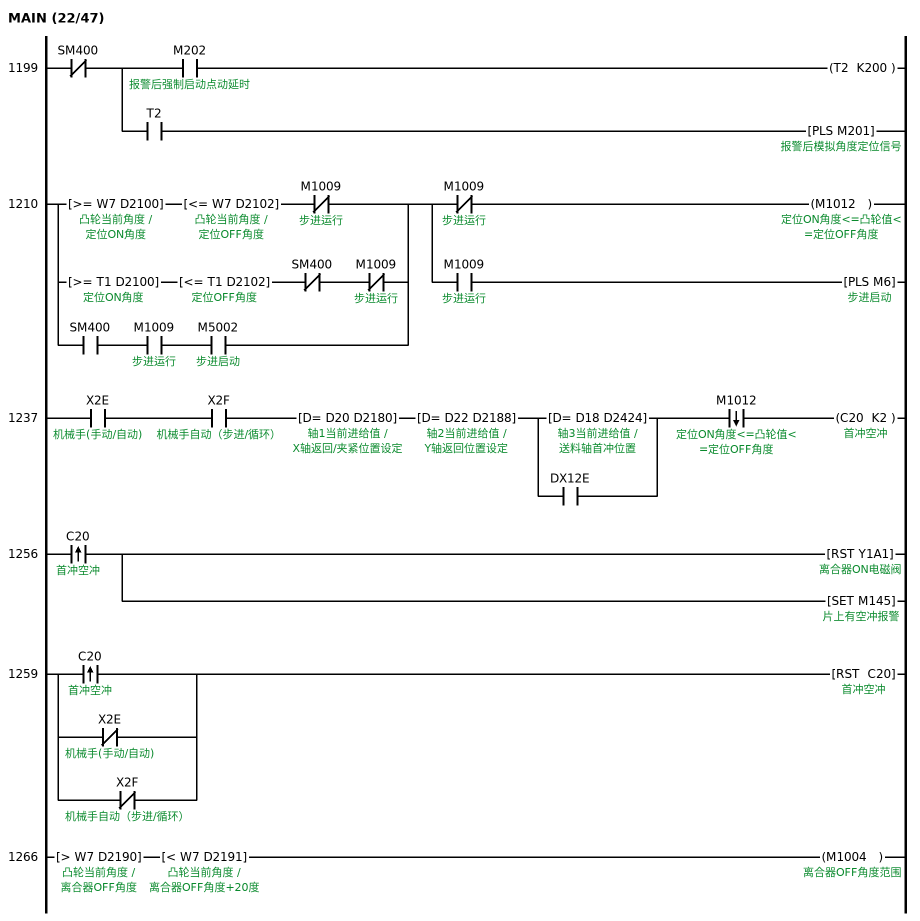
1199  LDI     SM400
      MPS
      AND     M202  ; 报警后强制启动点动延时
      OUT     T2 K200
      MPP
      AND     T2
      PLS     M201  ; 报警后模拟角度定位信号
1210  LD>=    W7 D2100  ; 凸轮当前角度 / 定位ON角度
      AND<=   W7 D2102  ; 凸轮当前角度 / 定位OFF角度
      ANI     M1009  ; 步进运行
      LD>=    T1 D2100  ; 定位ON角度
      AND<=   T1 D2102  ; 定位OFF角度
      ANI     SM400
      ANI     M1009  ; 步进运行
      ORB
      LD      SM400
      AND     M1009  ; 步进运行
      AND     M5002  ; 步进启动
      ORB
      MPS
      ANI     M1009  ; 步进运行
      OUT     M1012  ; 定位ON角度<=凸轮值<=定位OFF角度
      MPP
      AND     M1009  ; 步进运行
      PLS     M6  ; 步进启动
1237  LD      X2E  ; 机械手(手动/自动)
      AND     X2F  ; 机械手自动（步进/循环）
      ANDD=   D20 D2180  ; 轴1当前进给值 / X轴返回/夹紧位置设定
      ANDD=   D22 D2188  ; 轴2当前进给值 / Y轴返回位置设定
      LDD=    D18 D2424  ; 轴3当前进给值 / 送料轴首冲位置
      OR      DX12E
      ANB
      ANDF    M1012  ; 定位ON角度<=凸轮值<=定位OFF角度
      OUT     C20 K2  ; 首冲空冲
1256  LDP     C20  ; 首冲空冲
      RST     Y1A1  ; 离合器ON电磁阀
      SET     M145  ; 片上有空冲报警
1259  LDP     C20  ; 首冲空冲
      ORI     X2E  ; 机械手(手动/自动)
      ORI     X2F  ; 机械手自动（步进/循环）
      RST     C20  ; 首冲空冲
1266  LD>     W7 D2190  ; 凸轮当前角度 / 离合器OFF角度
      AND<    W7 D2191  ; 凸轮当前角度 / 离合器OFF角度+20度
      OUT     M1004  ; 离合器OFF角度范围
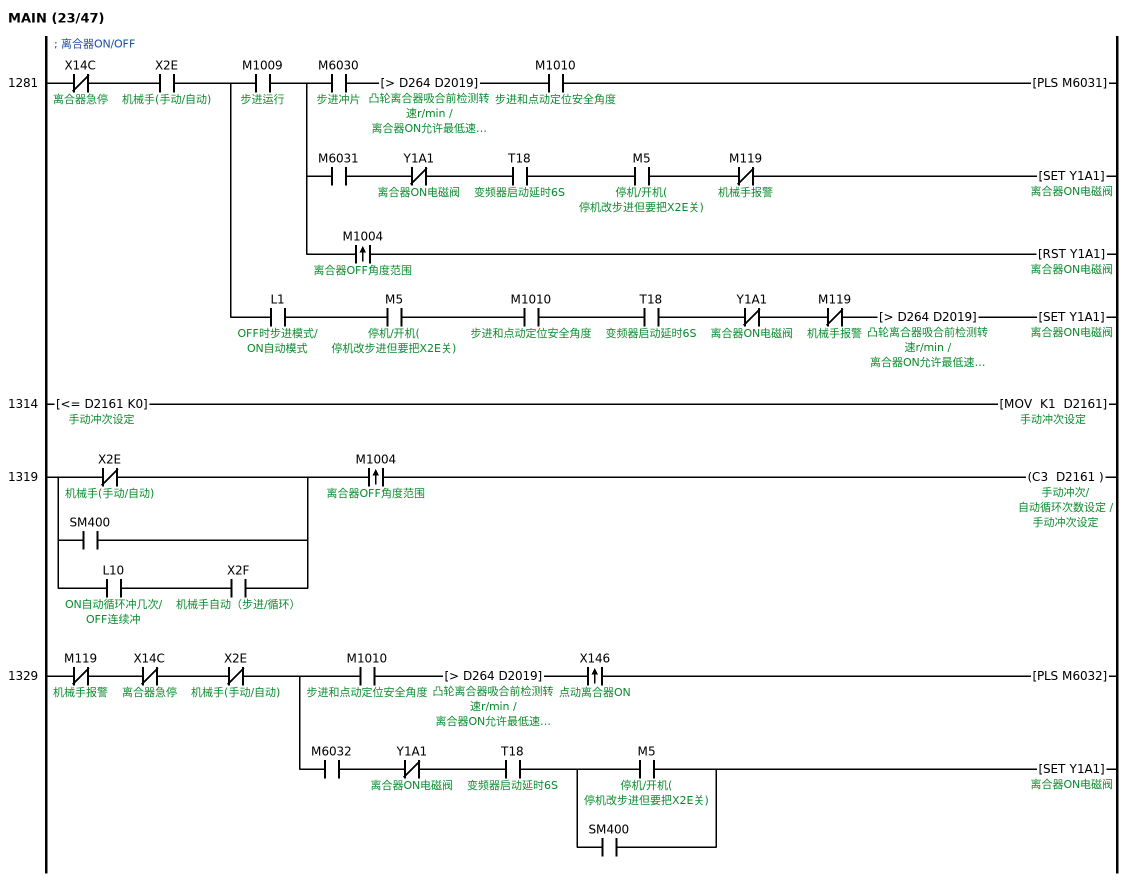
; 离合器ON/OFF
1281  LDI     X14C  ; 离合器急停
      AND     X2E  ; 机械手(手动/自动)
      MPS
      AND     M1009  ; 步进运行
      MPS
      AND     M6030  ; 步进冲片
      AND>    D264 D2019  ; 凸轮离合器吸合前检测转速r/min / 离合器ON允许最低速度设定
      AND     M1010  ; 步进和点动定位安全角度
      PLS     M6031
      MRD
      AND     M6031
      ANI     Y1A1  ; 离合器ON电磁阀
      AND     T18  ; 变频器启动延时6S
      AND     M5  ; 停机/开机(停机改步进但要把X2E关)
      ANI     M119  ; 机械手报警
      SET     Y1A1  ; 离合器ON电磁阀
      MPP
      ANDP    M1004  ; 离合器OFF角度范围
      RST     Y1A1  ; 离合器ON电磁阀
      MPP
      AND     L1  ; OFF时步进模式/ON自动模式
      AND     M5  ; 停机/开机(停机改步进但要把X2E关)
      AND     M1010  ; 步进和点动定位安全角度
      AND     T18  ; 变频器启动延时6S
      ANI     Y1A1  ; 离合器ON电磁阀
      ANI     M119  ; 机械手报警
      AND>    D264 D2019  ; 凸轮离合器吸合前检测转速r/min / 离合器ON允许最低速度设定
      SET     Y1A1  ; 离合器ON电磁阀
1314  LD<=    D2161 K0  ; 手动冲次设定
      MOV     K1 D2161
1319  LDI     X2E  ; 机械手(手动/自动)
      OR      SM400
      LD      L10  ; ON自动循环冲几次/OFF连续冲
      AND     X2F  ; 机械手自动（步进/循环）
      ORB
      ANDP    M1004  ; 离合器OFF角度范围
      OUT     C3 D2161  ; 手动冲次/自动循环次数设定 / 手动冲次设定
1329  LDI     M119  ; 机械手报警
      ANI     X14C  ; 离合器急停
      ANI     X2E  ; 机械手(手动/自动)
      MPS
      AND     M1010  ; 步进和点动定位安全角度
      AND>    D264 D2019  ; 凸轮离合器吸合前检测转速r/min / 离合器ON允许最低速度设定
      ANDP    X146  ; 点动离合器ON
      PLS     M6032
      MPP
      AND     M6032
      ANI     Y1A1  ; 离合器ON电磁阀
      AND     T18  ; 变频器启动延时6S
      LD      M5  ; 停机/开机(停机改步进但要把X2E关)
      OR      SM400
      ANB
      SET     Y1A1  ; 离合器ON电磁阀
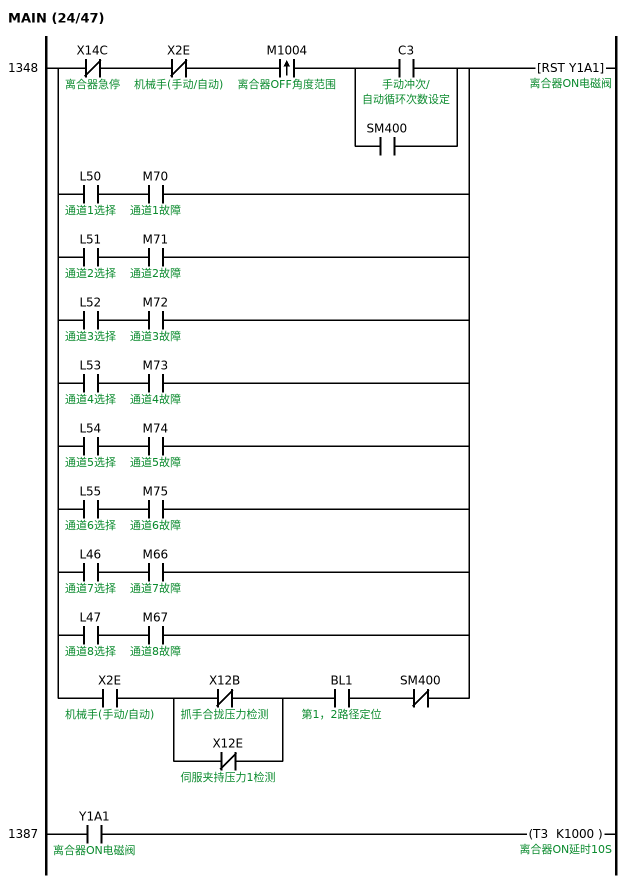
1348  LDI     X14C  ; 离合器急停
      ANI     X2E  ; 机械手(手动/自动)
      ANDP    M1004  ; 离合器OFF角度范围
      LD      C3  ; 手动冲次/自动循环次数设定
      OR      SM400
      ANB
      LD      L50  ; 通道1选择
      AND     M70  ; 通道1故障
      ORB
      LD      L51  ; 通道2选择
      AND     M71  ; 通道2故障
      ORB
      LD      L52  ; 通道3选择
      AND     M72  ; 通道3故障
      ORB
      LD      L53  ; 通道4选择
      AND     M73  ; 通道4故障
      ORB
      LD      L54  ; 通道5选择
      AND     M74  ; 通道5故障
      ORB
      LD      L55  ; 通道6选择
      AND     M75  ; 通道6故障
      ORB
      LD      L46  ; 通道7选择
      AND     M66  ; 通道7故障
      ORB
      LD      L47  ; 通道8选择
      AND     M67  ; 通道8故障
      ORB
      LD      X2E  ; 机械手(手动/自动)
      LDI     X12B  ; 抓手合拢压力检测
      ORI     X12E  ; 伺服夹持压力1检测
      ANB
      AND     BL1  ; 第1，2路径定位
      ANI     SM400
      ORB
      RST     Y1A1  ; 离合器ON电磁阀
1387  LD      Y1A1  ; 离合器ON电磁阀
      OUT     T3 K1000  ; 离合器ON延时10S
